// TIA Portal V17 export
// export: Created 2023-09-01T08:59:59.6540511Z, ExportSetting WithDefaults, DisplayName Totally Integrated Automation Portal, DisplayVersion V17 Update 6, DisplayName TIA Portal Openness, DisplayVersion V17 Update 6, DisplayName TIA Portal Teamcenter Gateway, DisplayVersion V17 Update 6, DisplayName TIA Portal Version Control Interface, DisplayVersion V17, DisplayName Simotion SCOUT TIA, DisplayVersion 5.4.3.0, DisplayName TIA Portal Test Suite Advanced, DisplayVersion V17 Update 1, DisplayName SIMOCODE ES, DisplayVersion V17 Update 5, DisplayName SINAMICS Startdrive Advanced, DisplayVersion V17 SP1, DisplayName SINAMICS Startdrive G130, G150, S120, S150, SINAMICS MV, S210, DisplayVersion V17 SP1, DisplayName SINAMICS Startdrive G110M, G120, G120C, G120D, G120P, G115D, DisplayVersion V17 SP1, DisplayName SIRIUS Safety ES, DisplayVersion V17 Update 5, DisplayName STEP 7 Professional, DisplayVersion V17 Update 6, DisplayName STEP 7 CFC, DisplayVersion V17 Update 1, DisplayName STEP 7 Safety, DisplayVersion V17 Update 6, DisplayName WinCC Advanced, DisplayVersion V17 Update 6, DisplayName SIMATIC Visualization Architect, DisplayVersion V17 Update 5
FUNCTION "03_Zone Cumulative" : Void   // FC4, F_FBD
{ S7_Optimized_Access := 'TRUE' }
VERSION : 0.1
// stored: AutoNumber true, IsIECCheckEnabled false, UDAEnableTagReadback false
BEGIN

REGION Network 1: S1 PB | ^SORTER UPPER COY =SC01
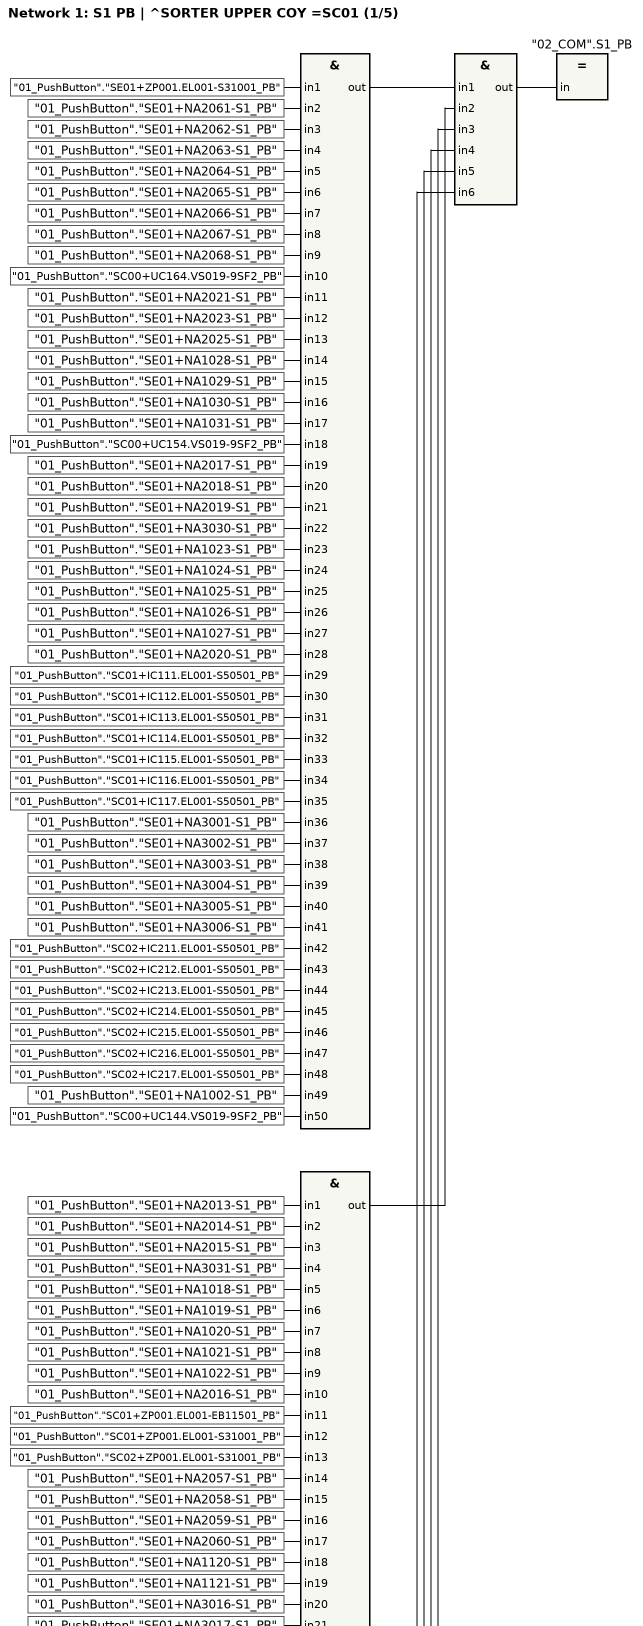
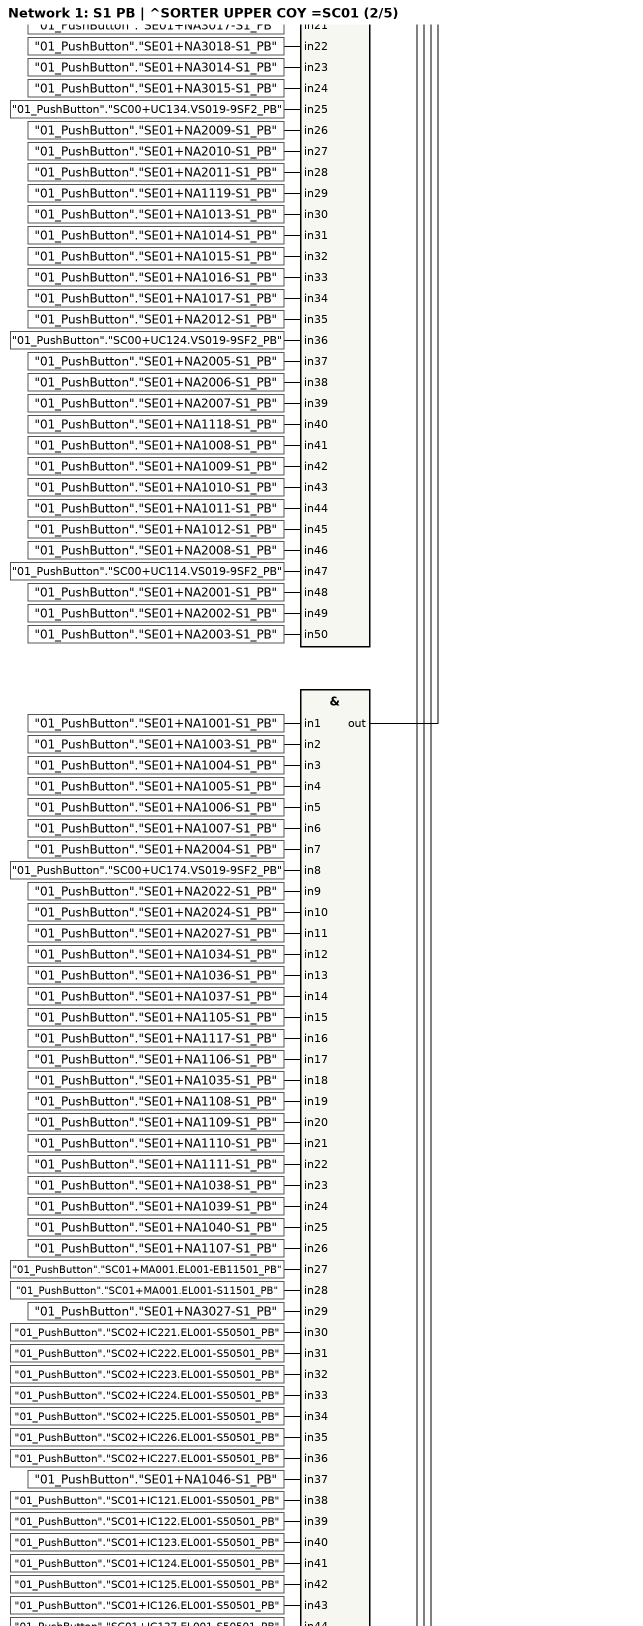
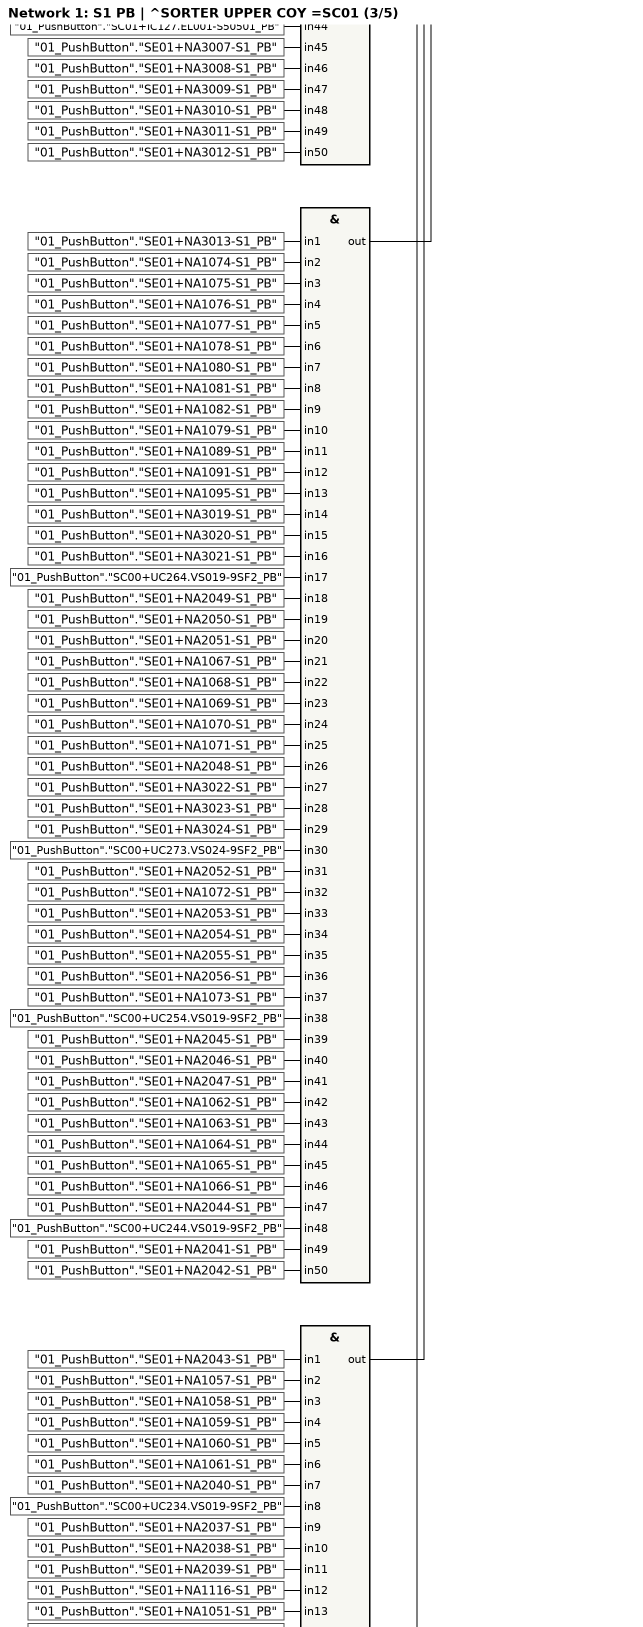
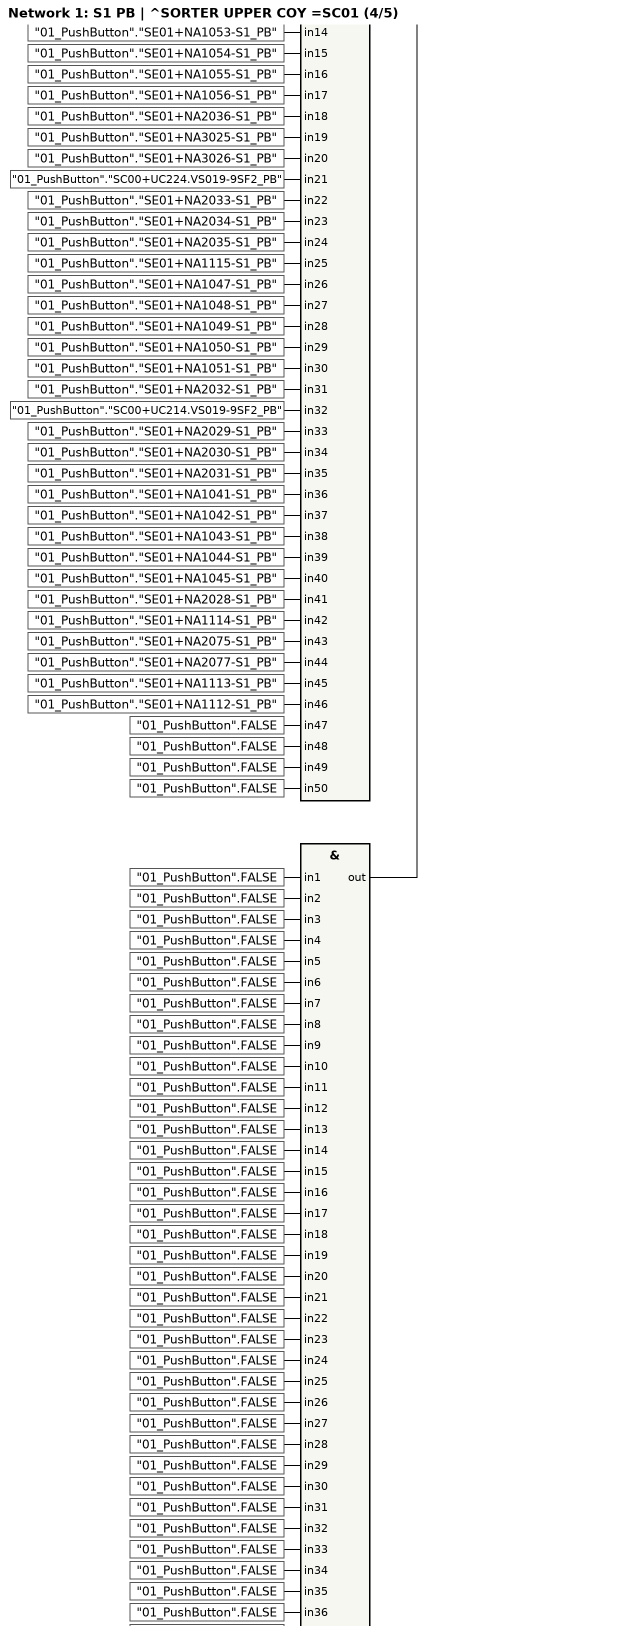
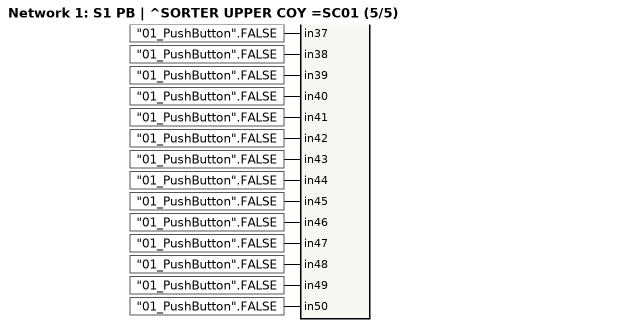
   "02_COM".S1_PB := "01_PushButton"."SE01+ZP001.EL001-S31001_PB" AND "01_PushButton"."SE01+NA2061-S1_PB" AND "01_PushButton"."SE01+NA2062-S1_PB" AND "01_PushButton"."SE01+NA2063-S1_PB" AND "01_PushButton"."SE01+NA2064-S1_PB" AND "01_PushButton"."SE01+NA2065-S1_PB" AND "01_PushButton"."SE01+NA2066-S1_PB" AND "01_PushButton"."SE01+NA2067-S1_PB" AND "01_PushButton"."SE01+NA2068-S1_PB" AND "01_PushButton"."SC00+UC164.VS019-9SF2_PB" AND "01_PushButton"."SE01+NA2021-S1_PB" AND "01_PushButton"."SE01+NA2023-S1_PB" AND "01_PushButton"."SE01+NA2025-S1_PB" AND "01_PushButton"."SE01+NA1028-S1_PB" AND "01_PushButton"."SE01+NA1029-S1_PB" AND "01_PushButton"."SE01+NA1030-S1_PB" AND "01_PushButton"."SE01+NA1031-S1_PB" AND "01_PushButton"."SC00+UC154.VS019-9SF2_PB" AND "01_PushButton"."SE01+NA2017-S1_PB" AND "01_PushButton"."SE01+NA2018-S1_PB" AND "01_PushButton"."SE01+NA2019-S1_PB" AND "01_PushButton"."SE01+NA3030-S1_PB" AND "01_PushButton"."SE01+NA1023-S1_PB" AND "01_PushButton"."SE01+NA1024-S1_PB" AND "01_PushButton"."SE01+NA1025-S1_PB" AND "01_PushButton"."SE01+NA1026-S1_PB" AND "01_PushButton"."SE01+NA1027-S1_PB" AND "01_PushButton"."SE01+NA2020-S1_PB" AND "01_PushButton"."SC01+IC111.EL001-S50501_PB" AND "01_PushButton"."SC01+IC112.EL001-S50501_PB" AND "01_PushButton"."SC01+IC113.EL001-S50501_PB" AND "01_PushButton"."SC01+IC114.EL001-S50501_PB" AND "01_PushButton"."SC01+IC115.EL001-S50501_PB" AND "01_PushButton"."SC01+IC116.EL001-S50501_PB" AND "01_PushButton"."SC01+IC117.EL001-S50501_PB" AND "01_PushButton"."SE01+NA3001-S1_PB" AND "01_PushButton"."SE01+NA3002-S1_PB" AND "01_PushButton"."SE01+NA3003-S1_PB" AND "01_PushButton"."SE01+NA3004-S1_PB" AND "01_PushButton"."SE01+NA3005-S1_PB" AND "01_PushButton"."SE01+NA3006-S1_PB" AND "01_PushButton"."SC02+IC211.EL001-S50501_PB" AND "01_PushButton"."SC02+IC212.EL001-S50501_PB" AND "01_PushButton"."SC02+IC213.EL001-S50501_PB" AND "01_PushButton"."SC02+IC214.EL001-S50501_PB" AND "01_PushButton"."SC02+IC215.EL001-S50501_PB" AND "01_PushButton"."SC02+IC216.EL001-S50501_PB" AND "01_PushButton"."SC02+IC217.EL001-S50501_PB" AND "01_PushButton"."SE01+NA1002-S1_PB" AND "01_PushButton"."SC00+UC144.VS019-9SF2_PB" AND "01_PushButton"."SE01+NA2013-S1_PB" AND "01_PushButton"."SE01+NA2014-S1_PB" AND "01_PushButton"."SE01+NA2015-S1_PB" AND "01_PushButton"."SE01+NA3031-S1_PB" AND "01_PushButton"."SE01+NA1018-S1_PB" AND "01_PushButton"."SE01+NA1019-S1_PB" AND "01_PushButton"."SE01+NA1020-S1_PB" AND "01_PushButton"."SE01+NA1021-S1_PB" AND "01_PushButton"."SE01+NA1022-S1_PB" AND "01_PushButton"."SE01+NA2016-S1_PB" AND "01_PushButton"."SC01+ZP001.EL001-EB11501_PB" AND "01_PushButton"."SC01+ZP001.EL001-S31001_PB" AND "01_PushButton"."SC02+ZP001.EL001-S31001_PB" AND "01_PushButton"."SE01+NA2057-S1_PB" AND "01_PushButton"."SE01+NA2058-S1_PB" AND "01_PushButton"."SE01+NA2059-S1_PB" AND "01_PushButton"."SE01+NA2060-S1_PB" AND "01_PushButton"."SE01+NA1120-S1_PB" AND "01_PushButton"."SE01+NA1121-S1_PB" AND "01_PushButton"."SE01+NA3016-S1_PB" AND "01_PushButton"."SE01+NA3017-S1_PB" AND "01_PushButton"."SE01+NA3018-S1_PB" AND "01_PushButton"."SE01+NA3014-S1_PB" AND "01_PushButton"."SE01+NA3015-S1_PB" AND "01_PushButton"."SC00+UC134.VS019-9SF2_PB" AND "01_PushButton"."SE01+NA2009-S1_PB" AND "01_PushButton"."SE01+NA2010-S1_PB" AND "01_PushButton"."SE01+NA2011-S1_PB" AND "01_PushButton"."SE01+NA1119-S1_PB" AND "01_PushButton"."SE01+NA1013-S1_PB" AND "01_PushButton"."SE01+NA1014-S1_PB" AND "01_PushButton"."SE01+NA1015-S1_PB" AND "01_PushButton"."SE01+NA1016-S1_PB" AND "01_PushButton"."SE01+NA1017-S1_PB" AND "01_PushButton"."SE01+NA2012-S1_PB" AND "01_PushButton"."SC00+UC124.VS019-9SF2_PB" AND "01_PushButton"."SE01+NA2005-S1_PB" AND "01_PushButton"."SE01+NA2006-S1_PB" AND "01_PushButton"."SE01+NA2007-S1_PB" AND "01_PushButton"."SE01+NA1118-S1_PB" AND "01_PushButton"."SE01+NA1008-S1_PB" AND "01_PushButton"."SE01+NA1009-S1_PB" AND "01_PushButton"."SE01+NA1010-S1_PB" AND "01_PushButton"."SE01+NA1011-S1_PB" AND "01_PushButton"."SE01+NA1012-S1_PB" AND "01_PushButton"."SE01+NA2008-S1_PB" AND "01_PushButton"."SC00+UC114.VS019-9SF2_PB" AND "01_PushButton"."SE01+NA2001-S1_PB" AND "01_PushButton"."SE01+NA2002-S1_PB" AND "01_PushButton"."SE01+NA2003-S1_PB" AND "01_PushButton"."SE01+NA1001-S1_PB" AND "01_PushButton"."SE01+NA1003-S1_PB" AND "01_PushButton"."SE01+NA1004-S1_PB" AND "01_PushButton"."SE01+NA1005-S1_PB" AND "01_PushButton"."SE01+NA1006-S1_PB" AND "01_PushButton"."SE01+NA1007-S1_PB" AND "01_PushButton"."SE01+NA2004-S1_PB" AND "01_PushButton"."SC00+UC174.VS019-9SF2_PB" AND "01_PushButton"."SE01+NA2022-S1_PB" AND "01_PushButton"."SE01+NA2024-S1_PB" AND "01_PushButton"."SE01+NA2027-S1_PB" AND "01_PushButton"."SE01+NA1034-S1_PB" AND "01_PushButton"."SE01+NA1036-S1_PB" AND "01_PushButton"."SE01+NA1037-S1_PB" AND "01_PushButton"."SE01+NA1105-S1_PB" AND "01_PushButton"."SE01+NA1117-S1_PB" AND "01_PushButton"."SE01+NA1106-S1_PB" AND "01_PushButton"."SE01+NA1035-S1_PB" AND "01_PushButton"."SE01+NA1108-S1_PB" AND "01_PushButton"."SE01+NA1109-S1_PB" AND "01_PushButton"."SE01+NA1110-S1_PB" AND "01_PushButton"."SE01+NA1111-S1_PB" AND "01_PushButton"."SE01+NA1038-S1_PB" AND "01_PushButton"."SE01+NA1039-S1_PB" AND "01_PushButton"."SE01+NA1040-S1_PB" AND "01_PushButton"."SE01+NA1107-S1_PB" AND "01_PushButton"."SC01+MA001.EL001-EB11501_PB" AND "01_PushButton"."SC01+MA001.EL001-S11501_PB" AND "01_PushButton"."SE01+NA3027-S1_PB" AND "01_PushButton"."SC02+IC221.EL001-S50501_PB" AND "01_PushButton"."SC02+IC222.EL001-S50501_PB" AND "01_PushButton"."SC02+IC223.EL001-S50501_PB" AND "01_PushButton"."SC02+IC224.EL001-S50501_PB" AND "01_PushButton"."SC02+IC225.EL001-S50501_PB" AND "01_PushButton"."SC02+IC226.EL001-S50501_PB" AND "01_PushButton"."SC02+IC227.EL001-S50501_PB" AND "01_PushButton"."SE01+NA1046-S1_PB" AND "01_PushButton"."SC01+IC121.EL001-S50501_PB" AND "01_PushButton"."SC01+IC122.EL001-S50501_PB" AND "01_PushButton"."SC01+IC123.EL001-S50501_PB" AND "01_PushButton"."SC01+IC124.EL001-S50501_PB" AND "01_PushButton"."SC01+IC125.EL001-S50501_PB" AND "01_PushButton"."SC01+IC126.EL001-S50501_PB" AND "01_PushButton"."SC01+IC127.EL001-S50501_PB" AND "01_PushButton"."SE01+NA3007-S1_PB" AND "01_PushButton"."SE01+NA3008-S1_PB" AND "01_PushButton"."SE01+NA3009-S1_PB" AND "01_PushButton"."SE01+NA3010-S1_PB" AND "01_PushButton"."SE01+NA3011-S1_PB" AND "01_PushButton"."SE01+NA3012-S1_PB" AND "01_PushButton"."SE01+NA3013-S1_PB" AND "01_PushButton"."SE01+NA1074-S1_PB" AND "01_PushButton"."SE01+NA1075-S1_PB" AND "01_PushButton"."SE01+NA1076-S1_PB" AND "01_PushButton"."SE01+NA1077-S1_PB" AND "01_PushButton"."SE01+NA1078-S1_PB" AND "01_PushButton"."SE01+NA1080-S1_PB" AND "01_PushButton"."SE01+NA1081-S1_PB" AND "01_PushButton"."SE01+NA1082-S1_PB" AND "01_PushButton"."SE01+NA1079-S1_PB" AND "01_PushButton"."SE01+NA1089-S1_PB" AND "01_PushButton"."SE01+NA1091-S1_PB" AND "01_PushButton"."SE01+NA1095-S1_PB" AND "01_PushButton"."SE01+NA3019-S1_PB" AND "01_PushButton"."SE01+NA3020-S1_PB" AND "01_PushButton"."SE01+NA3021-S1_PB" AND "01_PushButton"."SC00+UC264.VS019-9SF2_PB" AND "01_PushButton"."SE01+NA2049-S1_PB" AND "01_PushButton"."SE01+NA2050-S1_PB" AND "01_PushButton"."SE01+NA2051-S1_PB" AND "01_PushButton"."SE01+NA1067-S1_PB" AND "01_PushButton"."SE01+NA1068-S1_PB" AND "01_PushButton"."SE01+NA1069-S1_PB" AND "01_PushButton"."SE01+NA1070-S1_PB" AND "01_PushButton"."SE01+NA1071-S1_PB" AND "01_PushButton"."SE01+NA2048-S1_PB" AND "01_PushButton"."SE01+NA3022-S1_PB" AND "01_PushButton"."SE01+NA3023-S1_PB" AND "01_PushButton"."SE01+NA3024-S1_PB" AND "01_PushButton"."SC00+UC273.VS024-9SF2_PB" AND "01_PushButton"."SE01+NA2052-S1_PB" AND "01_PushButton"."SE01+NA1072-S1_PB" AND "01_PushButton"."SE01+NA2053-S1_PB" AND "01_PushButton"."SE01+NA2054-S1_PB" AND "01_PushButton"."SE01+NA2055-S1_PB" AND "01_PushButton"."SE01+NA2056-S1_PB" AND "01_PushButton"."SE01+NA1073-S1_PB" AND "01_PushButton"."SC00+UC254.VS019-9SF2_PB" AND "01_PushButton"."SE01+NA2045-S1_PB" AND "01_PushButton"."SE01+NA2046-S1_PB" AND "01_PushButton"."SE01+NA2047-S1_PB" AND "01_PushButton"."SE01+NA1062-S1_PB" AND "01_PushButton"."SE01+NA1063-S1_PB" AND "01_PushButton"."SE01+NA1064-S1_PB" AND "01_PushButton"."SE01+NA1065-S1_PB" AND "01_PushButton"."SE01+NA1066-S1_PB" AND "01_PushButton"."SE01+NA2044-S1_PB" AND "01_PushButton"."SC00+UC244.VS019-9SF2_PB" AND "01_PushButton"."SE01+NA2041-S1_PB" AND "01_PushButton"."SE01+NA2042-S1_PB" AND "01_PushButton"."SE01+NA2043-S1_PB" AND "01_PushButton"."SE01+NA1057-S1_PB" AND "01_PushButton"."SE01+NA1058-S1_PB" AND "01_PushButton"."SE01+NA1059-S1_PB" AND "01_PushButton"."SE01+NA1060-S1_PB" AND "01_PushButton"."SE01+NA1061-S1_PB" AND "01_PushButton"."SE01+NA2040-S1_PB" AND "01_PushButton"."SC00+UC234.VS019-9SF2_PB" AND "01_PushButton"."SE01+NA2037-S1_PB" AND "01_PushButton"."SE01+NA2038-S1_PB" AND "01_PushButton"."SE01+NA2039-S1_PB" AND "01_PushButton"."SE01+NA1116-S1_PB" AND "01_PushButton"."SE01+NA1051-S1_PB" AND "01_PushButton"."SE01+NA1053-S1_PB" AND "01_PushButton"."SE01+NA1054-S1_PB" AND "01_PushButton"."SE01+NA1055-S1_PB" AND "01_PushButton"."SE01+NA1056-S1_PB" AND "01_PushButton"."SE01+NA2036-S1_PB" AND "01_PushButton"."SE01+NA3025-S1_PB" AND "01_PushButton"."SE01+NA3026-S1_PB" AND "01_PushButton"."SC00+UC224.VS019-9SF2_PB" AND "01_PushButton"."SE01+NA2033-S1_PB" AND "01_PushButton"."SE01+NA2034-S1_PB" AND "01_PushButton"."SE01+NA2035-S1_PB" AND "01_PushButton"."SE01+NA1115-S1_PB" AND "01_PushButton"."SE01+NA1047-S1_PB" AND "01_PushButton"."SE01+NA1048-S1_PB" AND "01_PushButton"."SE01+NA1049-S1_PB" AND "01_PushButton"."SE01+NA1050-S1_PB" AND "01_PushButton"."SE01+NA1051-S1_PB" AND "01_PushButton"."SE01+NA2032-S1_PB" AND "01_PushButton"."SC00+UC214.VS019-9SF2_PB" AND "01_PushButton"."SE01+NA2029-S1_PB" AND "01_PushButton"."SE01+NA2030-S1_PB" AND "01_PushButton"."SE01+NA2031-S1_PB" AND "01_PushButton"."SE01+NA1041-S1_PB" AND "01_PushButton"."SE01+NA1042-S1_PB" AND "01_PushButton"."SE01+NA1043-S1_PB" AND "01_PushButton"."SE01+NA1044-S1_PB" AND "01_PushButton"."SE01+NA1045-S1_PB" AND "01_PushButton"."SE01+NA2028-S1_PB" AND "01_PushButton"."SE01+NA1114-S1_PB" AND "01_PushButton"."SE01+NA2075-S1_PB" AND "01_PushButton"."SE01+NA2077-S1_PB" AND "01_PushButton"."SE01+NA1113-S1_PB" AND "01_PushButton"."SE01+NA1112-S1_PB" AND "01_PushButton".FALSE AND "01_PushButton".FALSE AND "01_PushButton".FALSE AND "01_PushButton".FALSE AND "01_PushButton".FALSE AND "01_PushButton".FALSE AND "01_PushButton".FALSE AND "01_PushButton".FALSE AND "01_PushButton".FALSE AND "01_PushButton".FALSE AND "01_PushButton".FALSE AND "01_PushButton".FALSE AND "01_PushButton".FALSE AND "01_PushButton".FALSE AND "01_PushButton".FALSE AND "01_PushButton".FALSE AND "01_PushButton".FALSE AND "01_PushButton".FALSE AND "01_PushButton".FALSE AND "01_PushButton".FALSE AND "01_PushButton".FALSE AND "01_PushButton".FALSE AND "01_PushButton".FALSE AND "01_PushButton".FALSE AND "01_PushButton".FALSE AND "01_PushButton".FALSE AND "01_PushButton".FALSE AND "01_PushButton".FALSE AND "01_PushButton".FALSE AND "01_PushButton".FALSE AND "01_PushButton".FALSE AND "01_PushButton".FALSE AND "01_PushButton".FALSE AND "01_PushButton".FALSE AND "01_PushButton".FALSE AND "01_PushButton".FALSE AND "01_PushButton".FALSE AND "01_PushButton".FALSE AND "01_PushButton".FALSE AND "01_PushButton".FALSE AND "01_PushButton".FALSE AND "01_PushButton".FALSE AND "01_PushButton".FALSE AND "01_PushButton".FALSE AND "01_PushButton".FALSE AND "01_PushButton".FALSE AND "01_PushButton".FALSE AND "01_PushButton".FALSE AND "01_PushButton".FALSE AND "01_PushButton".FALSE AND "01_PushButton".FALSE AND "01_PushButton".FALSE AND "01_PushButton".FALSE AND "01_PushButton".FALSE;
END_REGION
END_FUNCTION
